// TIA Portal V17 export
// export: Created 2023-08-28T16:39:53.1884648Z, ExportSetting WithDefaults, DisplayName Totally Integrated Automation Portal, DisplayVersion V17 Update 5, DisplayName TIA Portal Openness, DisplayVersion V17 Update 5, DisplayName TIA Portal Teamcenter Gateway, DisplayVersion V17 Update 5, DisplayName TIA Portal Version Control Interface, DisplayVersion V17, DisplayName Simotion SCOUT TIA, DisplayVersion 5.4.3.0, DisplayName TIA Portal Test Suite Advanced, DisplayVersion V17 Update 1, DisplayName SIMOCODE ES, DisplayVersion V17 Update 5, DisplayName SINAMICS Startdrive Advanced, DisplayVersion V17 SP1, DisplayName SINAMICS Startdrive G130, G150, S120, S150, SINAMICS MV, S210, DisplayVersion V17 SP1, DisplayName SINAMICS Startdrive G110M, G120, G120C, G120D, G120P, G115D, DisplayVersion V17 SP1, DisplayName SIRIUS Safety ES, DisplayVersion V17 Update 5, DisplayName STEP 7 Professional, DisplayVersion V17 Update 5, DisplayName STEP 7 CFC, DisplayVersion V17 Update 1, DisplayName STEP 7 Safety, DisplayVersion V17, DisplayName WinCC Advanced, DisplayVersion V17 Update 5, DisplayName SIMATIC Visualization Architect, DisplayVersion V17 Update 5
FUNCTION "02_EM Push Button" : Void   // FC3, F_LAD
TITLE = Mirror PB
{ S7_Optimized_Access := 'TRUE' }
VERSION : 0.1
// stored: AutoNumber true, IsIECCheckEnabled false, UDAEnableTagReadback false
BEGIN

REGION Network 1: !!COLUMN_1$$
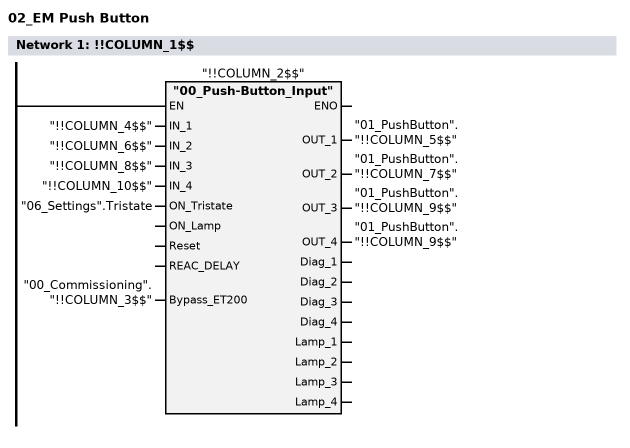
   RUNG wire#powerrail
      "!!COLUMN_2$$"(IN_1 := "!!COLUMN_4$$", IN_2 := "!!COLUMN_6$$", IN_3 := "!!COLUMN_8$$", IN_4 := "!!COLUMN_10$$", ON_Tristate := "06_Settings".Tristate, ON_Lamp :=, Reset :=, REAC_DELAY :=, Bypass_ET200 := "00_Commissioning"."!!COLUMN_3$$", OUT_1 => "01_PushButton"."!!COLUMN_5$$", OUT_2 => "01_PushButton"."!!COLUMN_7$$", OUT_3 => "01_PushButton"."!!COLUMN_9$$", OUT_4 => "01_PushButton"."!!COLUMN_9$$", Diag_1 =>, Diag_2 =>, Diag_3 =>, Diag_4 =>, Lamp_1 =>, Lamp_2 =>, Lamp_3 =>, Lamp_4 =>)
   END_RUNG
   // the same network as SCL:
   "!!COLUMN_2$$"(IN_1 := "!!COLUMN_4$$",   // "00_Push-Button_Input"
                  IN_2 := "!!COLUMN_6$$",
                  IN_3 := "!!COLUMN_8$$",
                  IN_4 := "!!COLUMN_10$$",
                  ON_Tristate := "06_Settings".Tristate,
                  Bypass_ET200 := "00_Commissioning"."!!COLUMN_3$$",
                  OUT_1 => "01_PushButton"."!!COLUMN_5$$",
                  OUT_2 => "01_PushButton"."!!COLUMN_7$$",
                  OUT_3 => "01_PushButton"."!!COLUMN_9$$",
                  OUT_4 => "01_PushButton"."!!COLUMN_9$$");
END_REGION
END_FUNCTION
